TYPE GearInMultiMaster_Statuses_typ :
	STRUCT
		InGear 			: 		BOOL;
		Busy 			: 		BOOL; 
		Active 			: 		BOOL; 
		CommandAborted 	: 		BOOL;
	END_STRUCT
END_TYPE

(* stored: Version 1.1.0.1, ProductVersion 3.1.4024.3
   DUT GearInMultiMaster_Statuses_typ: Id {ab7b6fd3-c4c8-0b04-1e57-574929e14933} *)
